# EPICS substitutions: TRITON/TRITON-IOC-01App/Db/TRITON_temp_channels.substitutions
file TRITON_temp_channels.template {

  pattern {PORT, P, CHAN, UID_COMMAND, IFFLNK}
  {"\$(PORT)", "\$(P)", "MC", "getChanUid(MC)", "#"}
  {"\$(PORT)", "\$(P)", "STIL", "getChanUid(STIL)", "#"}
  {"\$(PORT)", "\$(P)", "SORB", "getChanUid(SORB)", "#"}
  {"\$(PORT)", "\$(P)", "JTHX", "getChanUid(PT1)", "#"}
  {"\$(PORT)", "\$(P)", "4KHX", "getChanUid(PT2)", "#"}
  {"\$(PORT)", "\$(P)", "SAMPLE", "getSampleUid", ""}
}
